(* Logix 5000 project; controller TEC_81 vendor 1 type 14 code 148 rev 36.11; software revision 36.00; part 4 of 5 *)
(* tags used below, declared in another part *)
   FANUC : BOOL;
   Fanuc_Delta_Routine_Finish : BOOL;
   INICIO_FANUC : BOOL;
   Axis_1 : AXIS_CIP_DRIVE;
   Axis_2 : AXIS_CIP_DRIVE;   // Almacen 2
   Cmd_Axis_2 : BOOL;
   Cmd_Robot_Conv_1 : BOOL;
   Cmd_Robot_Conv_2 : BOOL;
   Cmd_YPickSafe_Alm1 : BOOL;
   Cmd_YPlaceSafe_Alm1 : BOOL;
   Cmd_YSafePos_Alm1 : BOOL;
   Cmd_YtoYOff_Alm1 : BOOL;
   Cmd_YtoYPick_Alm1 : BOOL;
   Cmd_YtoYPlace_Alm1 : BOOL;
   Cmd_YtoYPlaceOffset_Alm1 : BOOL;
   Consumeded_Signals_Conveyor_1_TEC_81 : DINT;
   Conveyor_1_Tomar_Pieza : BOOL;   // Señal del Conveyor 1 para Tomar Pieza Iniciar Ciclo
   Conveyor_2_Tomar_Pieza : BOOL;   // Señal del Conveyor 2 para Tomar Pieza Iniciar Ciclo
   EStops_OK : BOOL;   // E-Stop Close Loop Indicator
   EStops_OK_External : DINT;
   From_Robot : FromRobot_v02;
   From_Wh2 : DINT;
   FromStorage1 : DINT;
   Home_Sensor : BOOL;
   Interlocks_Ok : BOOL;   // Interlocks Close Loop Indicator
   LigthCurtain_ok : BOOL;   // Light Curtains Close Loop Indicator
   MC_1_EStop : DCI_STOP;   // Status of E-Stop 1
   MC_1_EStop_Status : BOOL;   // General status of inputs
   MC_1_LigthCurtain : DCI_STOP;   // Status of Light Curtain 1
   MC_2_EStop : DCI_STOP;   // Status of E-Stop 2
   MC_2_EStop_Status : BOOL;   // General status of inputs
   MC_3_EStop : DCI_STOP;   // Status of E-Stop 3
   MC_3_EStop_Status : BOOL;   // General status of inputs
   MC_4_EStop : DCI_STOP;   // Status of E-Stop 4
   MC_4_EStop_Status : BOOL;   // General status of inputs
   MC_5_EStop : DCI_STOP;   // Status of E-Stop 5
   MC_5_EStop_Status : BOOL;   // General status of inputs
   MEMORIA_DELTA_INICIO : BOOL;   // Inicio de delta
   ok : BOOL;
   Ons : INT;
   Operation_Mode : BOOL;   // Operation Mode for HMI (1) Manual (0) Automatico
   Paro_Emergencia_Almacen_1 : BOOL;   // Stopping signal of Torc Off Almacen 1
   Paro_Emergencia_Almacen_2 : BOOL;   // Stopping signal of Torc Off Almacen 2
   Produced_Signals_TEC_81_Conveyor_1 : DINT;
   Retorno_Pieza_A_Conveyor_1 : BOOL;
   Robot_Step : DINT;
   Safety_FromTEC81 : Safety;
   Signal_Fanuc_Tomar_Pieza_Conv_1 : BOOL;   // Señal para Tomar pieza desde el Conveyor 1 Hacia CNC
   Storage_1_Y_ActualPosition : REAL;
   Storage_2_Y_ActualPosition : REAL;
   Tec81_to_Wh2 : DINT;
   Test : BOOL;
   test_com : BOOL;   // bit e comunicacion
   TOF_STO_KinetixStorage2 : TIMER;
   TT : BOOL;
(* MainProgram, continued *)

ROUTINE _10_ExternalComm   (* ladder *)
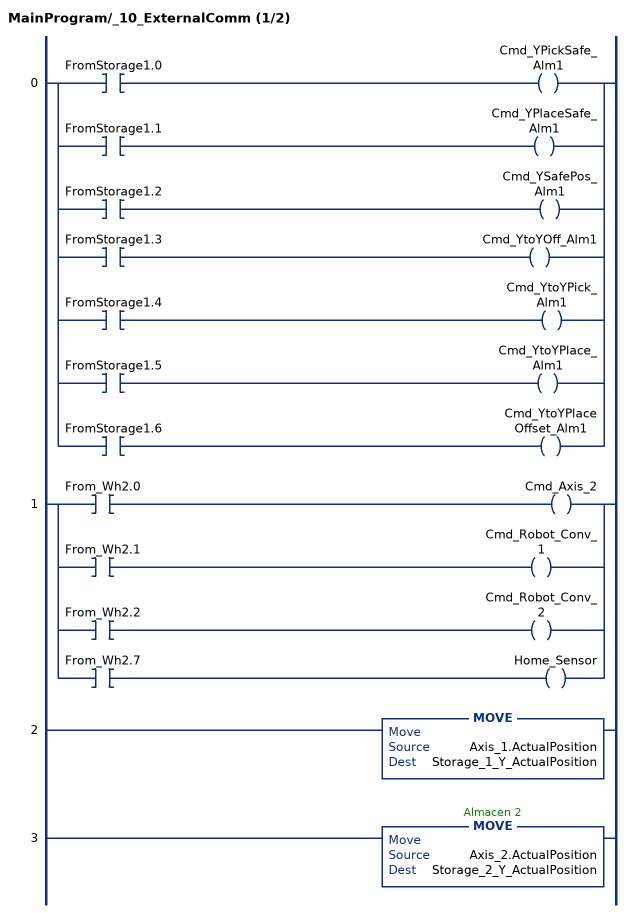
   0: [XIC(FromStorage1.0) OTE(Cmd_YPickSafe_Alm1) ,XIC(FromStorage1.1) OTE(Cmd_YPlaceSafe_Alm1) ,XIC(FromStorage1.2) OTE(Cmd_YSafePos_Alm1) ,XIC(FromStorage1.3) OTE(Cmd_YtoYOff_Alm1) ,XIC(FromStorage1.4) OTE(Cmd_YtoYPick_Alm1) ,XIC(FromStorage1.5) OTE(Cmd_YtoYPlace_Alm1) ,XIC(FromStorage1.6) OTE(Cmd_YtoYPlaceOffset_Alm1) ];
   1: [XIC(From_Wh2.0) OTE(Cmd_Axis_2) ,XIC(From_Wh2.1) OTE(Cmd_Robot_Conv_1) ,XIC(From_Wh2.2) OTE(Cmd_Robot_Conv_2) ,XIC(From_Wh2.7) OTE(Home_Sensor) ];
   2: MOVE(Axis_1.ActualPosition,Storage_1_Y_ActualPosition);
   3: MOVE(Axis_2.ActualPosition,Storage_2_Y_ActualPosition);
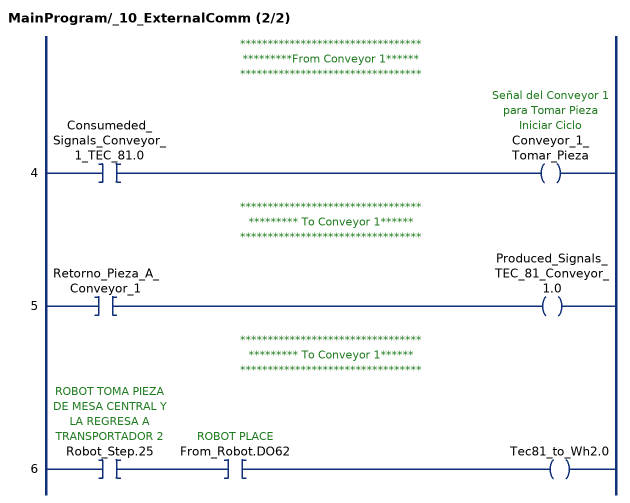
   // *********************************
   // *********From Conveyor 1******
   // *********************************
   4: XIC(Consumeded_Signals_Conveyor_1_TEC_81.0)OTE(Conveyor_1_Tomar_Pieza);
   // *********************************
   // ********* To Conveyor 1******
   // *********************************
   5: XIC(Retorno_Pieza_A_Conveyor_1)OTE(Produced_Signals_TEC_81_Conveyor_1.0);
   // *********************************
   // ********* To Conveyor 1******
   // *********************************
   6: XIC(Robot_Step.25)XIC(From_Robot.DO62)OTE(Tec81_to_Wh2.0);
END_ROUTINE

ROUTINE _11_External   (* ladder *)
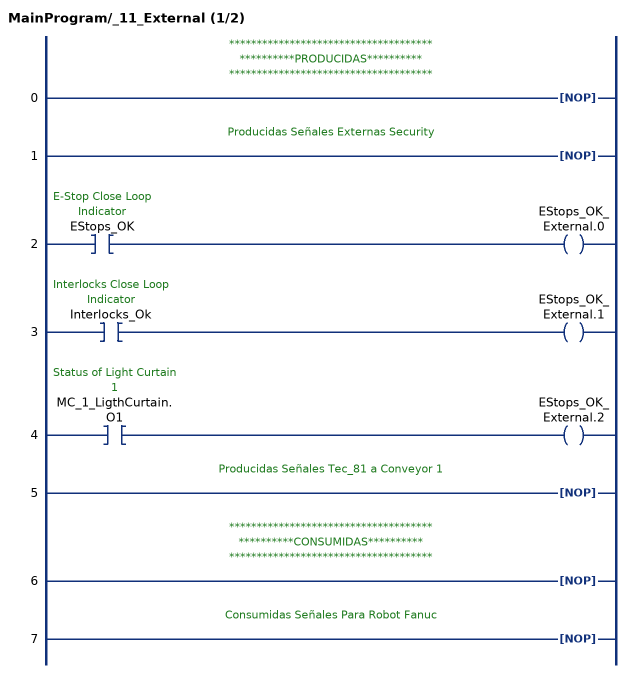
   // *************************************
   // **********PRODUCIDAS**********
   // *************************************
   0: NOP();
   // Producidas Señales Externas Security
   1: NOP();
   2: XIC(EStops_OK)OTE(EStops_OK_External.0);
   3: XIC(Interlocks_Ok)OTE(EStops_OK_External.1);
   4: XIC(MC_1_LigthCurtain.O1)OTE(EStops_OK_External.2);
   // Producidas Señales Tec_81 a Conveyor 1
   5: NOP();
   // *************************************
   // **********CONSUMIDAS**********
   // *************************************
   6: NOP();
   // Consumidas Señales Para Robot Fanuc
   7: NOP();
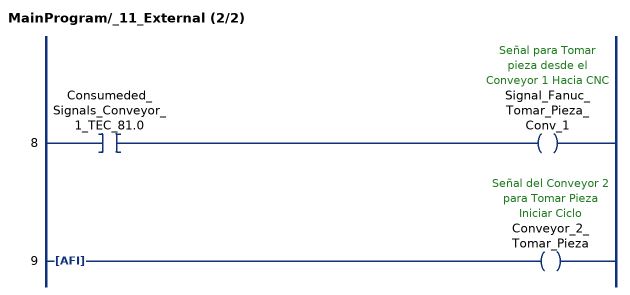
   8: XIC(Consumeded_Signals_Conveyor_1_TEC_81.0)OTE(Signal_Fanuc_Tomar_Pieza_Conv_1);
   9: AFI()OTE(Conveyor_2_Tomar_Pieza);
END_ROUTINE

ROUTINE CNC1   (* ladder *)
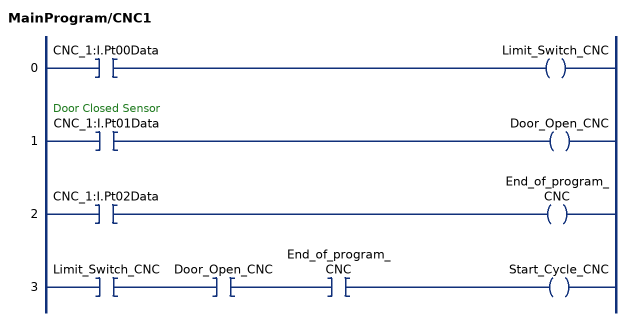
   0: XIC(CNC_1:I.Pt00Data)OTE(Limit_Switch_CNC);
   1: XIC(CNC_1:I.Pt01Data)OTE(Door_Open_CNC);
   2: XIC(CNC_1:I.Pt02Data)OTE(End_of_program_CNC);
   3: XIC(Limit_Switch_CNC)XIC(Door_Open_CNC)XIC(End_of_program_CNC)OTE(Start_Cycle_CNC);
END_ROUTINE

ROUTINE FANUC   (* ladder *)
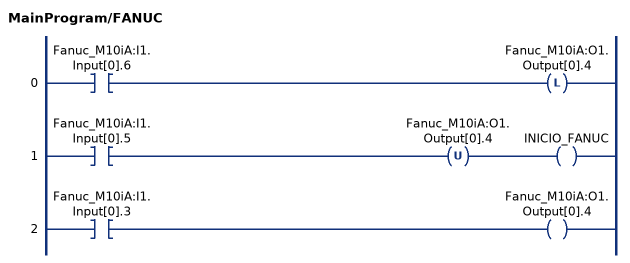
   0: XIC(Fanuc_M10iA:I1.Input[0].6)OTL(Fanuc_M10iA:O1.Output[0].4);
   1: XIC(Fanuc_M10iA:I1.Input[0].5)OTU(Fanuc_M10iA:O1.Output[0].4)OTE(INICIO_FANUC);
   2: XIC(Fanuc_M10iA:I1.Input[0].3)OTE(Fanuc_M10iA:O1.Output[0].4);
END_ROUTINE

ROUTINE Fanuc_Delta   (* ladder *)
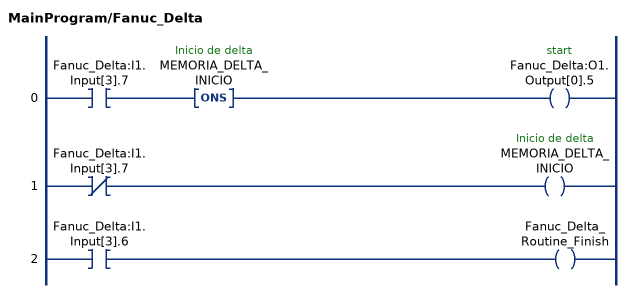
   0: XIC(Fanuc_Delta:I1.Input[3].7)ONS(MEMORIA_DELTA_INICIO)OTE(Fanuc_Delta:O1.Output[0].5);
   1: XIO(Fanuc_Delta:I1.Input[3].7)OTE(MEMORIA_DELTA_INICIO);
   2: XIC(Fanuc_Delta:I1.Input[3].6)OTE(Fanuc_Delta_Routine_Finish);
END_ROUTINE

ROUTINE MainRoutine   (* ladder *)
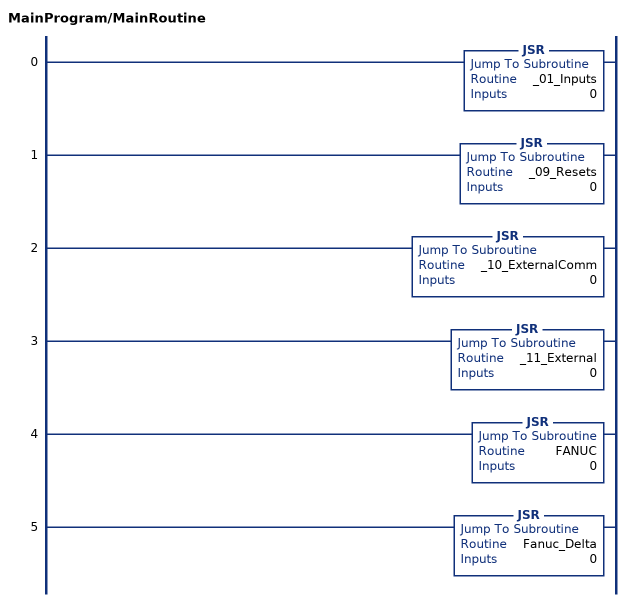
   0: JSR(_01_Inputs,0);
   1: JSR(_09_Resets,0);
   2: JSR(_10_ExternalComm,0);
   3: JSR(_11_External,0);
   4: JSR(FANUC,0);
   5: JSR(Fanuc_Delta,0);
END_ROUTINE
END_PROGRAM

PROGRAM Manu_camaras
END_PROGRAM

PROGRAM SafetyProgram   (* main routine MainRoutine, safety *)
VAR
   Close_CNC_Door : BOOL;
   Close_pneumatic_press : BOOL;
   Door_Open_CNC : BOOL;
   dummy : BOOL;
   End_of_program_CNC : BOOL;
   Fanuc_Place_CNC : BOOL;
   Lasers_OK : BOOL;   // Laser Scanner Close Loop Indicator
   Limit_Switch_CNC : BOOL;
   LS_1 : DCI_STOP := (InputStatus := 1, RestartType := 1, ColdStartType := 1, SafetyFunction := 1, DiscrepancyTime := 200);   // Status of Laser Scanner 1
   LS_1_Status : BOOL := 1;   // General status of inputs
   LS_2 : DCI_STOP := (InputStatus := 1, RestartType := 1, ColdStartType := 1, SafetyFunction := 1, DiscrepancyTime := 200);   // Status of Laser Scanner 2
   LS_2_Status : BOOL := 1;   // General status of inputs
   Mat_1 : DCI_STOP := (ChannelA := 1, InputStatus := 1, RestartType := 1, ColdStartType := 1, SafetyFunction := 4, DiscrepancyTime := 200, FP := 1, FaultCode := 32);   // Status of Safety Mat 1
   Mat_1_Status : BOOL;   // General status of inputs
   ONS_Laser_1 : BOOL;   // One time execution for reset
   ONS_Laser_2 : BOOL;   // One time execution for reset
   ONS_Mat_1 : BOOL;   // One time execution for reset
   Open_pneumatic_press : BOOL;
   Output_Enable_Laser_1 : BOOL;   // General status of Laser 1
   Output_Enable_Laser_2 : BOOL;   // General status of Laser 2
   Output_Enable_Mat_1 : BOOL;   // General status of Mat 1
   Safety_Close_Loop_ok : BOOL := 1;   // General Safety Indicator
   Safety_Latch_Timer : TIMER := (PRE := 500);
   Safety_Mat_ok : BOOL;   // Safety Mat Close Loop Indicator
   Safety_Reset_General : BOOL;   // Unified General Reset
   Start_CNC_Routine : BOOL;
   Start_Cycle_CNC : BOOL;
   Stop_routine_CNC : BOOL;
   T_prepare : TIMER := (PRE := 3000);
   T_stop : TIMER := (PRE := 1000);
   test_1 : BOOL;
   test_21 : BOOL;
   Timer_Cyc_start : TIMER := (PRE := 5000);
   TOF_STO_KinetixStorage1 : TIMER := (PRE := 10000, EN := 1, DN := 1);
END_VAR

ROUTINE Almacenes   (* ladder *)
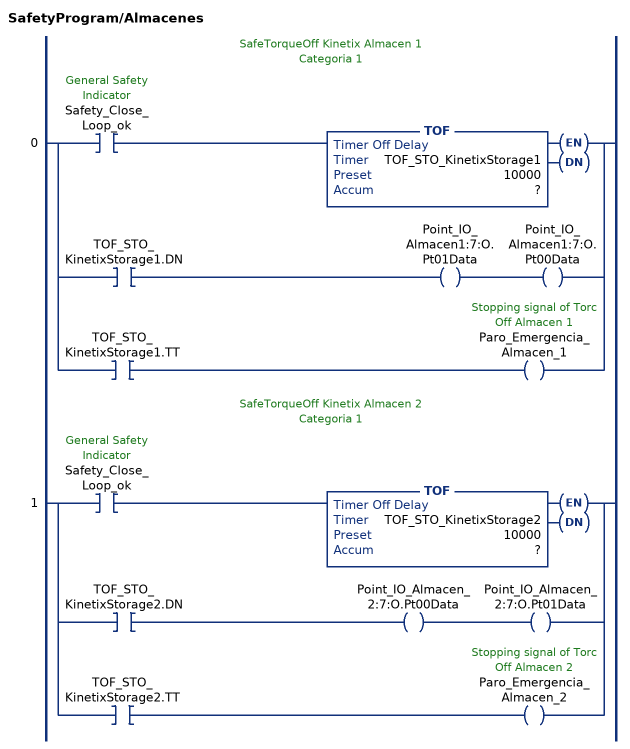
   // SafeTorqueOff Kinetix Almacen 1
   // Categoria 1
   0: [XIC(Safety_Close_Loop_ok) TOF(TOF_STO_KinetixStorage1,?,?) ,XIC(TOF_STO_KinetixStorage1.DN) OTE(Point_IO_Almacen1:7:O.Pt01Data) OTE(Point_IO_Almacen1:7:O.Pt00Data) ,XIC(TOF_STO_KinetixStorage1.TT) OTE(Paro_Emergencia_Almacen_1) ];
   // SafeTorqueOff Kinetix Almacen 2
   // Categoria 1
   1: [XIC(Safety_Close_Loop_ok) TOF(TOF_STO_KinetixStorage2,?,?) ,XIC(TOF_STO_KinetixStorage2.DN) OTE(Point_IO_Almacen_2:7:O.Pt00Data) OTE(Point_IO_Almacen_2:7:O.Pt01Data) ,XIC(TOF_STO_KinetixStorage2.TT) OTE(Paro_Emergencia_Almacen_2) ];
END_ROUTINE

ROUTINE CNC_routine   (* ladder *)
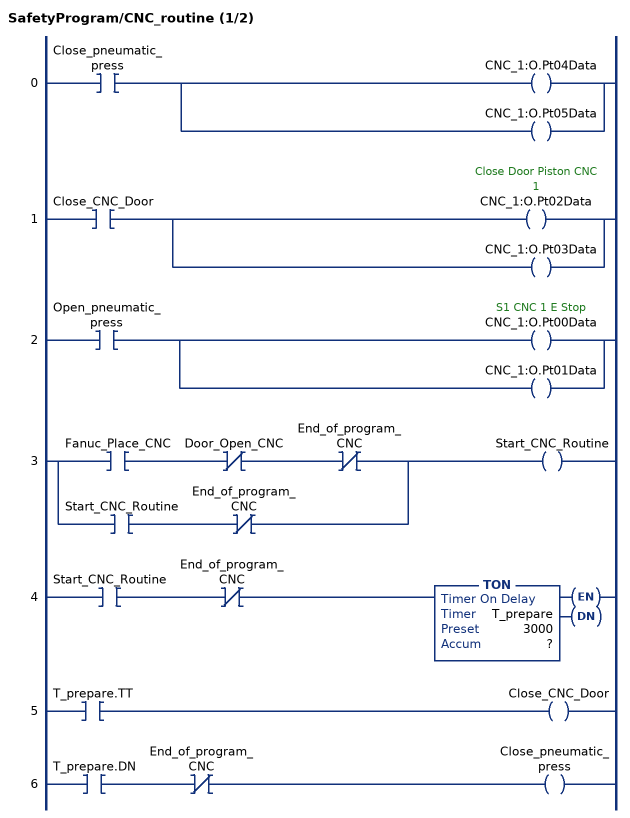
   0: XIC(Close_pneumatic_press)[OTE(CNC_1:O.Pt04Data) ,OTE(CNC_1:O.Pt05Data) ];
   1: XIC(Close_CNC_Door)[OTE(CNC_1:O.Pt02Data) ,OTE(CNC_1:O.Pt03Data) ];
   2: XIC(Open_pneumatic_press)[OTE(CNC_1:O.Pt00Data) ,OTE(CNC_1:O.Pt01Data) ];
   3: [XIC(Fanuc_Place_CNC) XIO(Door_Open_CNC) XIO(End_of_program_CNC) ,XIC(Start_CNC_Routine) XIO(End_of_program_CNC) ]OTE(Start_CNC_Routine);
   4: XIC(Start_CNC_Routine)XIO(End_of_program_CNC)TON(T_prepare,?,?);
   5: XIC(T_prepare.TT)OTE(Close_CNC_Door);
   6: XIC(T_prepare.DN)XIO(End_of_program_CNC)OTE(Close_pneumatic_press);
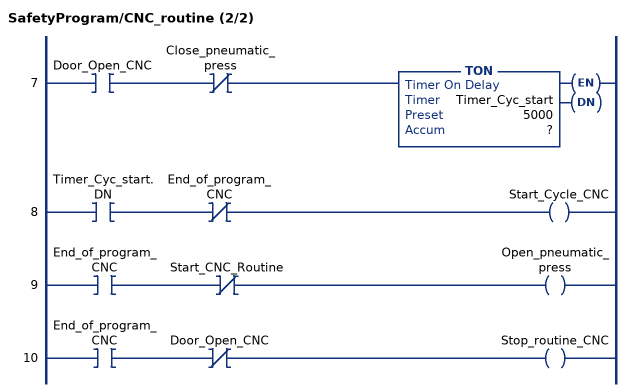
   7: XIC(Door_Open_CNC)XIO(Close_pneumatic_press)TON(Timer_Cyc_start,?,?);
   8: XIC(Timer_Cyc_start.DN)XIO(End_of_program_CNC)OTE(Start_Cycle_CNC);
   9: XIC(End_of_program_CNC)XIO(Start_CNC_Routine)OTE(Open_pneumatic_press);
   10: XIC(End_of_program_CNC)XIO(Door_Open_CNC)OTE(Stop_routine_CNC);
END_ROUTINE

ROUTINE Conveyors   (* ladder *)
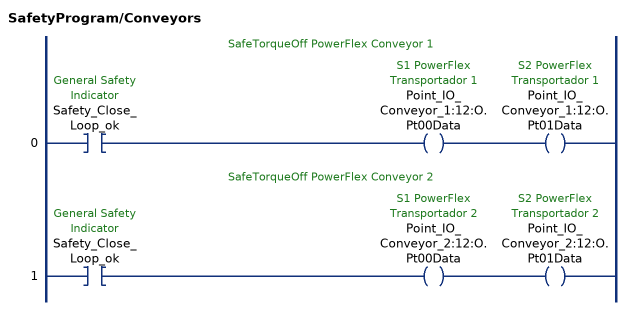
   // SafeTorqueOff PowerFlex Conveyor 1
   0: XIC(Safety_Close_Loop_ok)OTE(Point_IO_Conveyor_1:12:O.Pt00Data)OTE(Point_IO_Conveyor_1:12:O.Pt01Data);
   // SafeTorqueOff PowerFlex Conveyor 2
   1: XIC(Safety_Close_Loop_ok)OTE(Point_IO_Conveyor_2:12:O.Pt00Data)OTE(Point_IO_Conveyor_2:12:O.Pt01Data);
END_ROUTINE

ROUTINE Estops   (* ladder *)
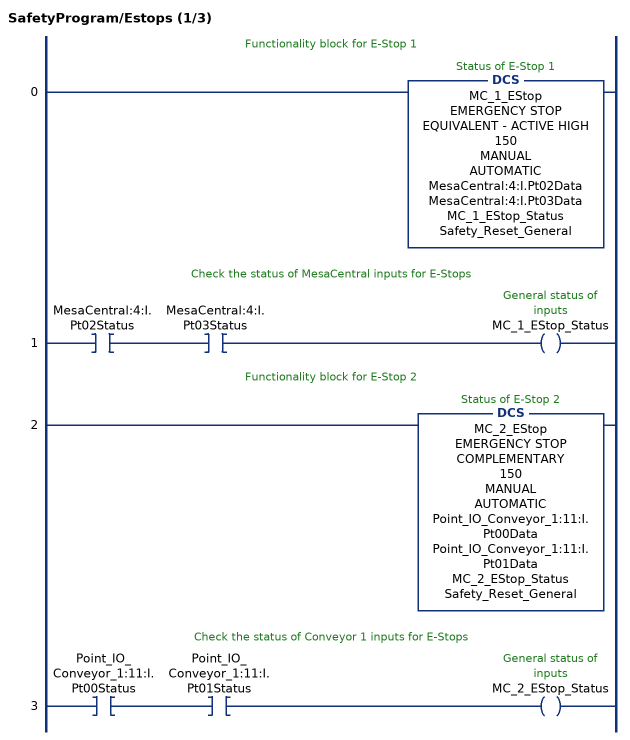
   // Functionality block for E-Stop 1
   0: DCS(MC_1_EStop,EMERGENCY STOP,EQUIVALENT - ACTIVE HIGH,150,MANUAL,AUTOMATIC,MesaCentral:4:I.Pt02Data,MesaCentral:4:I.Pt03Data,MC_1_EStop_Status,Safety_Reset_General);
   // Check the status of MesaCentral inputs for E-Stops
   1: XIC(MesaCentral:4:I.Pt02Status)XIC(MesaCentral:4:I.Pt03Status)OTE(MC_1_EStop_Status);
   // Functionality block for E-Stop 2
   2: DCS(MC_2_EStop,EMERGENCY STOP,COMPLEMENTARY,150,MANUAL,AUTOMATIC,Point_IO_Conveyor_1:11:I.Pt00Data,Point_IO_Conveyor_1:11:I.Pt01Data,MC_2_EStop_Status,Safety_Reset_General);
   // Check the status of Conveyor 1 inputs for E-Stops
   3: XIC(Point_IO_Conveyor_1:11:I.Pt00Status)XIC(Point_IO_Conveyor_1:11:I.Pt01Status)OTE(MC_2_EStop_Status);
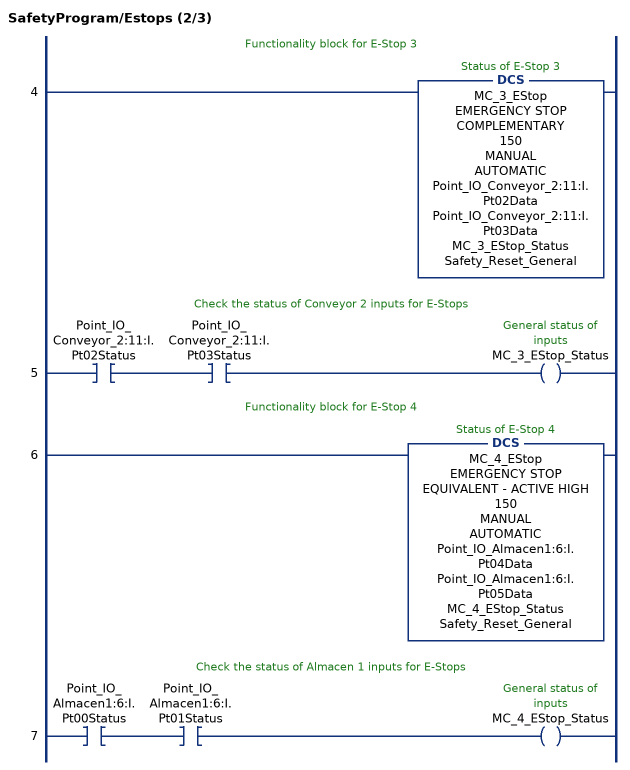
   // Functionality block for E-Stop 3
   4: DCS(MC_3_EStop,EMERGENCY STOP,COMPLEMENTARY,150,MANUAL,AUTOMATIC,Point_IO_Conveyor_2:11:I.Pt02Data,Point_IO_Conveyor_2:11:I.Pt03Data,MC_3_EStop_Status,Safety_Reset_General);
   // Check the status of Conveyor 2 inputs for E-Stops
   5: XIC(Point_IO_Conveyor_2:11:I.Pt02Status)XIC(Point_IO_Conveyor_2:11:I.Pt03Status)OTE(MC_3_EStop_Status);
   // Functionality block for E-Stop 4
   6: DCS(MC_4_EStop,EMERGENCY STOP,EQUIVALENT - ACTIVE HIGH,150,MANUAL,AUTOMATIC,Point_IO_Almacen1:6:I.Pt04Data,Point_IO_Almacen1:6:I.Pt05Data,MC_4_EStop_Status,Safety_Reset_General);
   // Check the status of Almacen 1 inputs for E-Stops
   7: XIC(Point_IO_Almacen1:6:I.Pt00Status)XIC(Point_IO_Almacen1:6:I.Pt01Status)OTE(MC_4_EStop_Status);
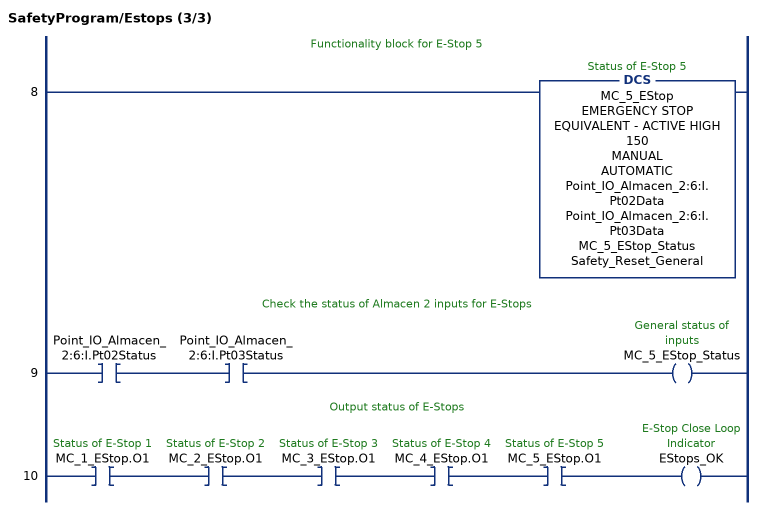
   // Functionality block for E-Stop 5
   8: DCS(MC_5_EStop,EMERGENCY STOP,EQUIVALENT - ACTIVE HIGH,150,MANUAL,AUTOMATIC,Point_IO_Almacen_2:6:I.Pt02Data,Point_IO_Almacen_2:6:I.Pt03Data,MC_5_EStop_Status,Safety_Reset_General);
   // Check the status of Almacen 2 inputs for E-Stops
   9: XIC(Point_IO_Almacen_2:6:I.Pt02Status)XIC(Point_IO_Almacen_2:6:I.Pt03Status)OTE(MC_5_EStop_Status);
   // Output status of E-Stops
   10: XIC(MC_1_EStop.O1)XIC(MC_2_EStop.O1)XIC(MC_3_EStop.O1)XIC(MC_4_EStop.O1)XIC(MC_5_EStop.O1)OTE(EStops_OK);
END_ROUTINE

ROUTINE External_COMM   (* ladder *)
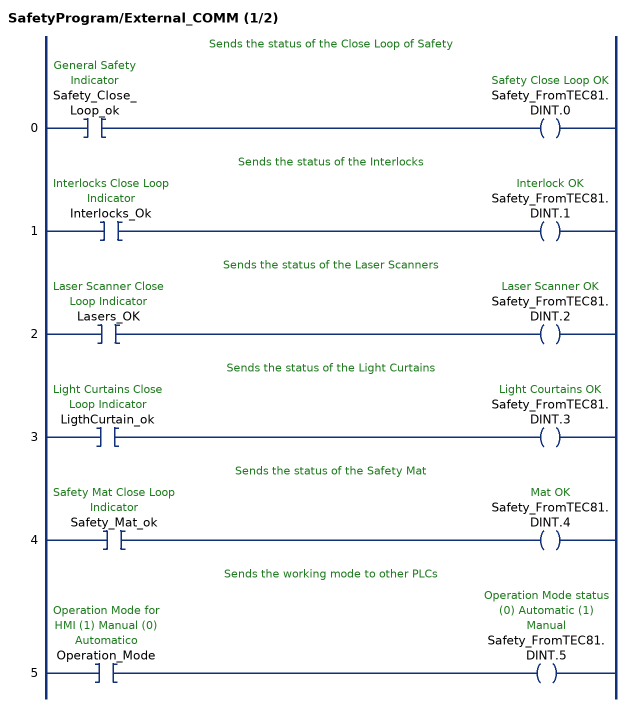
   // Sends the status of the Close Loop of Safety
   0: XIC(Safety_Close_Loop_ok)OTE(Safety_FromTEC81.DINT.0);
   // Sends the status of the Interlocks
   1: XIC(Interlocks_Ok)OTE(Safety_FromTEC81.DINT.1);
   // Sends the status of the Laser Scanners
   2: XIC(Lasers_OK)OTE(Safety_FromTEC81.DINT.2);
   // Sends the status of the Light Curtains
   3: XIC(LigthCurtain_ok)OTE(Safety_FromTEC81.DINT.3);
   // Sends the status of the Safety Mat
   4: XIC(Safety_Mat_ok)OTE(Safety_FromTEC81.DINT.4);
   // Sends the working mode to other PLCs
   5: XIC(Operation_Mode)OTE(Safety_FromTEC81.DINT.5);
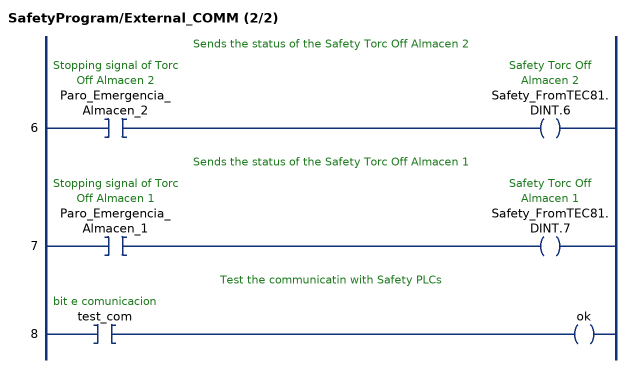
   // Sends the status of the Safety Torc Off Almacen 2
   6: XIC(Paro_Emergencia_Almacen_2)OTE(Safety_FromTEC81.DINT.6);
   // Sends the status of the Safety Torc Off Almacen 1
   7: XIC(Paro_Emergencia_Almacen_1)OTE(Safety_FromTEC81.DINT.7);
   // Test the communicatin with Safety PLCs
   8: XIC(test_com)OTE(ok);
END_ROUTINE

ROUTINE Fanuc_Delta   (* ladder *)
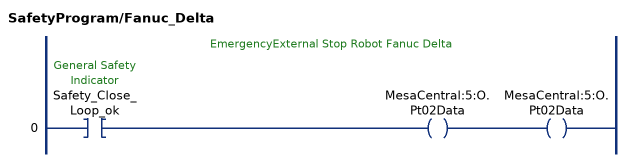
   // EmergencyExternal Stop Robot Fanuc Delta
   0: XIC(Safety_Close_Loop_ok)OTE(MesaCentral:5:O.Pt02Data)OTE(MesaCentral:5:O.Pt02Data);
END_ROUTINE
